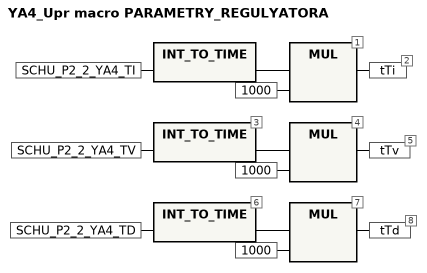
[picture p530: YA4_Upr macro PARAMETRY_REGULYATORA (CFC)]
_CFC_ (* Continuous Function Chart, elements in execution order *)
#0 MACRO PARAMETRY_REGULYATORA()
	#1 INT_TO_TIME(SCHU_P2_2_YA4_TI)
	#2 MUL(#1, 1000)
	#3 tTi <= #2
	#4 INT_TO_TIME(SCHU_P2_2_YA4_TV)
	#5 MUL(#4, 1000)
	#6 tTv <= #5
	#7 INT_TO_TIME(SCHU_P2_2_YA4_TD)
	#8 MUL(#7, 1000)
	#9 tTd <= #8
END_MACRO
#10 SEL(SCHU_P2_2_SA6_DI7_A, 0, #15.out 1)
#11 AND(SCHU_P2_2_UE3_T_DOST, NOT SCHU_P2_2_Z_OTKAZ_VTORICH_SEP, SCHU_P2_2_SA6_DI7_A, SCHU_P2_2_UST_RE_RABOTA)
#12 SEL(#11, eHVACCtrlMode_Manual, eHVACCtrlMode_Auto)
#13 OR(SCHU_P2_2_Z_OTKAZ_VTORICH_SEP, NOT SCHU_P2_2_UST_RE_RABOTA)
#14 SEL(#13, SCHU_P2_2_YA4_UP_VN, 0)
#15 YA4_PID:FB_HVACPIDCtrl(eHVACDataSecurityType_Idle, FALSE, TRUE, SCHU_P2_2_UE3_T_UST, SCHU_P2_2_UE3_T_VN, tTaskCycleTime, tTaskCycleTime, #12, #14, #14, FALSE, SCHU_P2_2_SB, deadRange, direction, SCHU_P2_2_YA4_KP, tTi, tTv, tTd, rYMin, rYMax)
#16 SCHU_P2_2_YA4_ZAD_VN <= #10
#17 SCHU_P2_2_YA4_RASSOG <= #15.out 2
#18 SUB(#10, SCHU_P2_2_YA4_UP_VN)
#19 SCHU_P2_2_YA4_RASSOG_POL <= #18
_END_CFC_
END_PROGRAM

(* POU IM/razr_pusk, CFC *)
PROGRAM razr_pusk
VAR
END_VAR
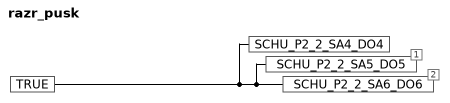
_CFC_ (* Continuous Function Chart, elements in execution order *)
#0 SCHU_P2_2_SA4_DO4 <= TRUE
#1 SCHU_P2_2_SA5_DO5 <= TRUE
#2 SCHU_P2_2_SA6_DO6 <= TRUE
_END_CFC_
(* the same logic as Structured Text *)
SCHU_P2_2_SA4_DO4 := TRUE;
SCHU_P2_2_SA5_DO5 := TRUE;
SCHU_P2_2_SA6_DO6 := TRUE;
END_PROGRAM

(* POU Output/ALL_Output, CFC *)
PROGRAM ALL_Output
VAR
END_VAR
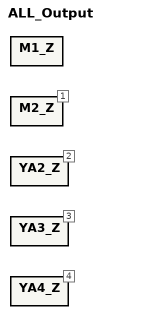
_CFC_ (* Continuous Function Chart, elements in execution order *)
#0 M1_Z()
#1 M2_Z()
#2 YA2_Z()
#3 YA3_Z()
#4 YA4_Z()
_END_CFC_
(* the same logic as Structured Text *)
M1_Z();
M2_Z();
YA2_Z();
YA3_Z();
YA4_Z();
END_PROGRAM

(* POU Output/AO/M1_Z, CFC *)
PROGRAM M1_Z
VAR
	fb_HVACAO_SCHU_P2_2_UZ1_AO1: FB_HVACAnalogOutput;
	enableFeedbCtrl: BOOL := FALSE;
	hysFbCtrl: REAL := 0;
	direction: BOOL;
	delay: TIME := T#0s;
	hi: REAL := 50;
	low: REAL := 0;

END_VAR
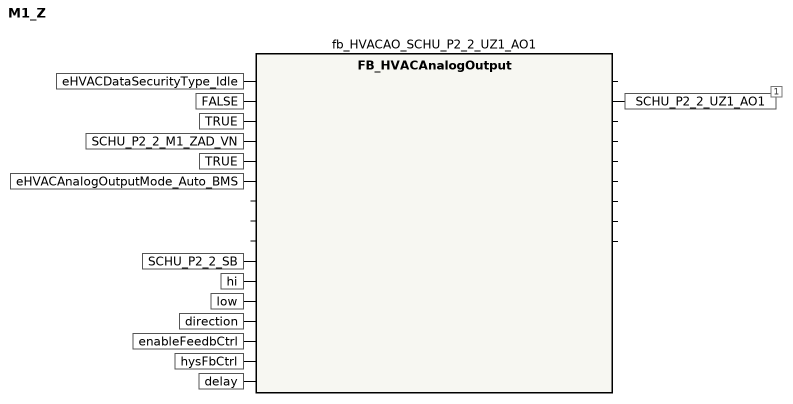
_CFC_ (* Continuous Function Chart, elements in execution order *)
#0 fb_HVACAO_SCHU_P2_2_UZ1_AO1:FB_HVACAnalogOutput(eHVACDataSecurityType_Idle, FALSE, TRUE, SCHU_P2_2_M1_ZAD_VN, TRUE, eHVACAnalogOutputMode_Auto_BMS, -, -, -, SCHU_P2_2_SB, hi, low, direction, enableFeedbCtrl, hysFbCtrl, delay)
#1 SCHU_P2_2_UZ1_AO1 <= #0.out 2
_END_CFC_
END_PROGRAM

(* POU Output/AO/M2_Z, CFC *)
PROGRAM M2_Z
VAR
	fb_HVACAO_SCHU_P2_2_UZ2_AO5: FB_HVACAnalogOutput;
	enableFeedbCtrl: BOOL := FALSE;
	hysFbCtrl: REAL := 0;
	direction: BOOL;
	delay: TIME := T#0s;
	hi: REAL := 50;
	low: REAL := 0;
END_VAR
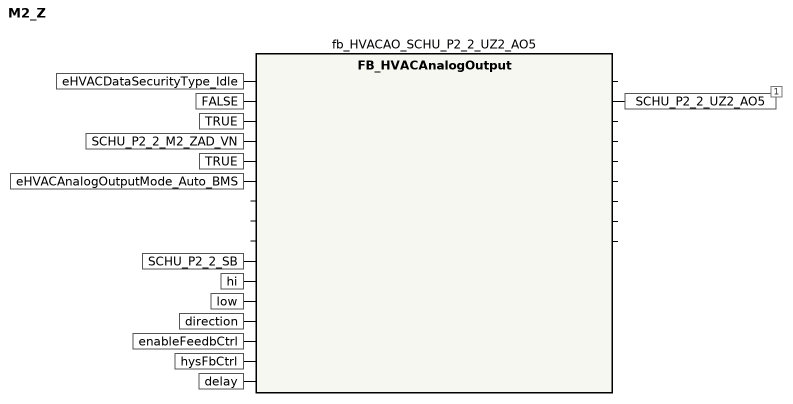
_CFC_ (* Continuous Function Chart, elements in execution order *)
#0 fb_HVACAO_SCHU_P2_2_UZ2_AO5:FB_HVACAnalogOutput(eHVACDataSecurityType_Idle, FALSE, TRUE, SCHU_P2_2_M2_ZAD_VN, TRUE, eHVACAnalogOutputMode_Auto_BMS, -, -, -, SCHU_P2_2_SB, hi, low, direction, enableFeedbCtrl, hysFbCtrl, delay)
#1 SCHU_P2_2_UZ2_AO5 <= #0.out 2
_END_CFC_
END_PROGRAM

(* POU Output/AO/YA2_Z, CFC *)
PROGRAM YA2_Z
VAR
	fb_HVACAO_SCHU_P2_2_YA2_AO2: FB_HVACAnalogOutput;
	enableFeedbCtrl: BOOL := FALSE;
	hysFbCtrl: REAL := 0;
	direction: BOOL;
	delay: TIME := T#0s;
END_VAR
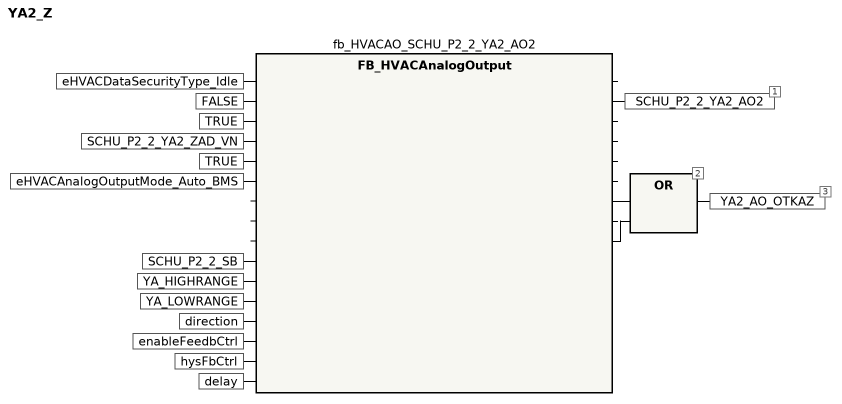
_CFC_ (* Continuous Function Chart, elements in execution order *)
#0 fb_HVACAO_SCHU_P2_2_YA2_AO2:FB_HVACAnalogOutput(eHVACDataSecurityType_Idle, FALSE, TRUE, SCHU_P2_2_YA2_ZAD_VN, TRUE, eHVACAnalogOutputMode_Auto_BMS, -, -, -, SCHU_P2_2_SB, YA_HIGHRANGE, YA_LOWRANGE, direction, enableFeedbCtrl, hysFbCtrl, delay)
#1 SCHU_P2_2_YA2_AO2 <= #0.out 2
#2 OR(#0.out 7, #0.out 9)
#3 YA2_AO_OTKAZ <= #2
_END_CFC_
END_PROGRAM

(* POU Output/AO/YA3_Z, CFC *)
PROGRAM YA3_Z
VAR
	fb_HVACAO_SCHU_P2_2_YA3_AO3: FB_HVACAnalogOutput;
	enableFeedbCtrl: BOOL := FALSE;
	hysFbCtrl: REAL := 0;
	direction: BOOL;
	delay: TIME := T#0s;
END_VAR
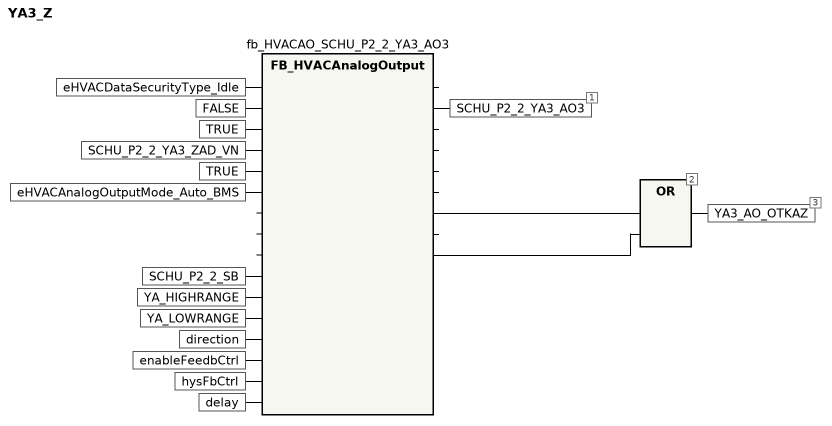
_CFC_ (* Continuous Function Chart, elements in execution order *)
#0 fb_HVACAO_SCHU_P2_2_YA3_AO3:FB_HVACAnalogOutput(eHVACDataSecurityType_Idle, FALSE, TRUE, SCHU_P2_2_YA3_ZAD_VN, TRUE, eHVACAnalogOutputMode_Auto_BMS, -, -, -, SCHU_P2_2_SB, YA_HIGHRANGE, YA_LOWRANGE, direction, enableFeedbCtrl, hysFbCtrl, delay)
#1 SCHU_P2_2_YA3_AO3 <= #0.out 2
#2 OR(#0.out 7, #0.out 9)
#3 YA3_AO_OTKAZ <= #2
_END_CFC_
END_PROGRAM

(* POU Output/AO/YA4_Z, CFC *)
PROGRAM YA4_Z
VAR
	fb_HVACAO_SCHU_P2_2_YA4_AO4: FB_HVACAnalogOutput;
	enableFeedbCtrl: BOOL := FALSE;
	hysFbCtrl: REAL := 0;
	direction: BOOL;
	delay: TIME := T#0s;
END_VAR
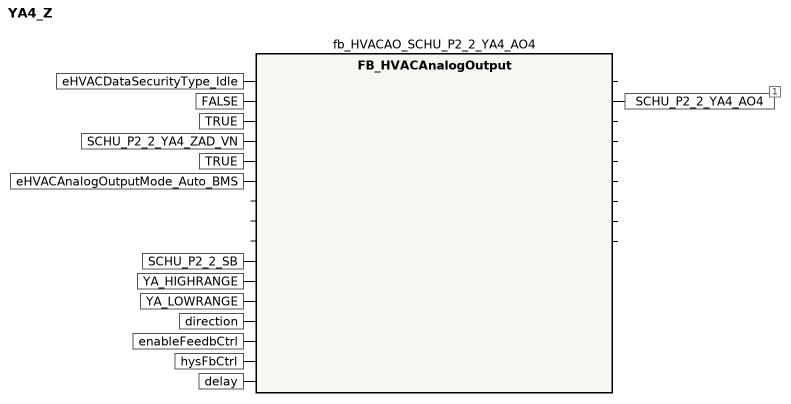
_CFC_ (* Continuous Function Chart, elements in execution order *)
#0 fb_HVACAO_SCHU_P2_2_YA4_AO4:FB_HVACAnalogOutput(eHVACDataSecurityType_Idle, FALSE, TRUE, SCHU_P2_2_YA4_ZAD_VN, TRUE, eHVACAnalogOutputMode_Auto_BMS, -, -, -, SCHU_P2_2_SB, YA_HIGHRANGE, YA_LOWRANGE, direction, enableFeedbCtrl, hysFbCtrl, delay)
#1 SCHU_P2_2_YA4_AO4 <= #0.out 2
_END_CFC_
END_PROGRAM

(* POU Input/ModBus/MB_UZT, CFC *)
PROGRAM MB_UZT
VAR
	MB_READ_REGS: ModbusRtuMaster_KL6x22B;
	Quantity: WORD:= 4;
	MBAddr: WORD:= 16#3000;
	Error: BOOL;
	Errorld: MODBUS_ERRORS;
	cbRead: UINT;

	TON1: TON;

	UnitID_2: BYTE:=2;
	rs_s: RS;
	UnitID_1: BYTE := 1;

	SWT: BOOL;
	ton2: TON;
	tp1: TOF;

END_VAR
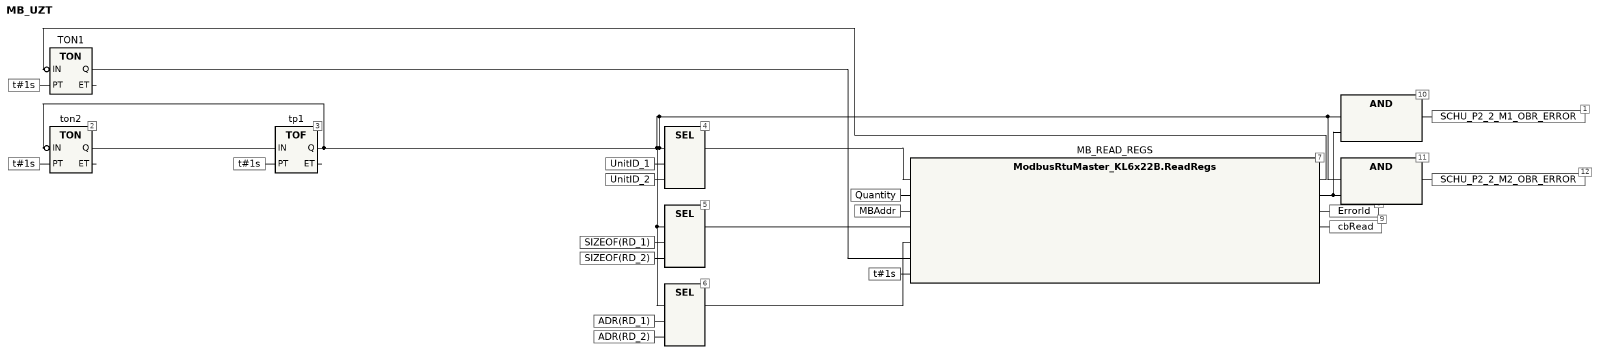
_CFC_ (* Continuous Function Chart, elements in execution order *)
#0 TON1:TON(IN: NOT #7.out 1, PT: t#1s)
#1 SCHU_P2_2_M1_OBR_ERROR <= #10
#2 ton2:TON(IN: NOT #3.Q, PT: t#1s)
#3 tp1:TOF(IN: #2.Q, PT: t#1s)
#4 SEL(#3.Q, UnitID_1, UnitID_2)
#5 SEL(#3.Q, SIZEOF(RD_1), SIZEOF(RD_2))
#6 SEL(#3.Q, ADR(RD_1), ADR(RD_2))
#7 MB_READ_REGS:ModbusRtuMaster_KL6x22B.ReadRegs(#4, Quantity, MBAddr, #5, #6, #0.Q, t#1s)
#8 Errorld <= #7.out 3
#9 cbRead <= #7.out 4
#10 AND(#3.Q, #7.out 2)
#11 AND(#3.Q, #7.out 2)
#12 SCHU_P2_2_M2_OBR_ERROR <= #11
_END_CFC_
END_PROGRAM

(* POU Input/AI/UE1_VL, CFC *)
PROGRAM UE1_VL
VAR
	fb_UE2_VL: ISTOK_ANALOGVH;
	ofset: REAL;
	fb_UE2_VLbUST: ISTOK_GT;
END_VAR
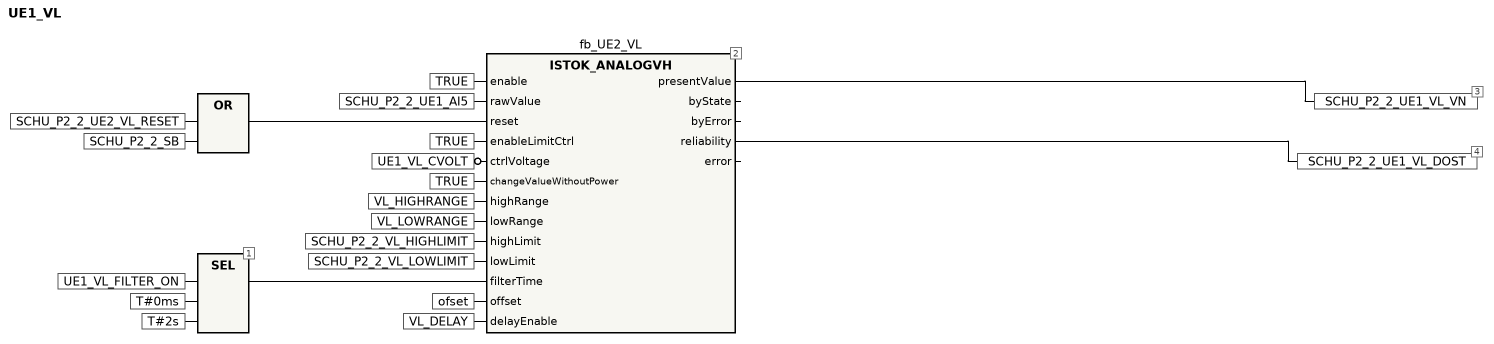
